// TIA Portal V17 export
// export: Created 2022-07-20T07:02:34.5888701Z, ExportSetting WithDefaults, DisplayName Totally Integrated Automation Portal, DisplayVersion V17, DisplayName TIA Portal Openness, DisplayVersion V17, DisplayName TIA Portal Version Control Interface, DisplayVersion V17, DisplayName SINAMICS Startdrive Advanced, DisplayVersion V17, DisplayName SINAMICS Startdrive G130, G150, S120, S150, SINAMICS MV, S210, DisplayVersion V17, DisplayName SINAMICS Startdrive G110M, G120, G120C, G120D, G120P, G115D, DisplayVersion V17, DisplayName STEP 7 Professional, DisplayVersion V17, DisplayName STEP 7 Safety, DisplayVersion V17, DisplayName WinCC Advanced, DisplayVersion V17
FUNCTION_BLOCK "FB10373_IOLinkConfig_Any"   // FB10373, LAD
{ S7_Optimized_Access := 'TRUE' }
VERSION : 0.1
// stored: AutoNumber false, IsIECCheckEnabled false, IsRetainMemResEnabled false, MemoryReserve 100, SetENOAutomatically false, UDAEnableTagReadback false
   VAR_INPUT
      Ackowledge : Bool;
      PortDevice : Int;
      Id : HW_IO;
      RequestGetParamID : Bool;
      RequestSetParamID : Bool;
      Index : Int;
      SubIndex : Int;
      Length : Int;
   END_VAR
   VAR_OUTPUT
      ParamIdDone : Bool;
      ParamConfigFault : Array[0..231] of Byte;
      Error : Bool;
      Status : Word;
   END_VAR
   VAR_IN_OUT
      Value : Array[0..231] of Byte;
   END_VAR
   VAR
      CommandStruct : Struct
         In : Struct
            TrigStart_Pulse : Bool;
            Id : HW_IO;
            rw : Bool;
            Port : Int;
            index : Int;
            subindex : Int;
            length : Int;
         END_STRUCT;
         Out : Struct
            Done : Bool;
            busy : Bool;
            Error : Bool;
            Status : Word;
         END_STRUCT;
         InOut : Struct
            Data : Array[0..231] of Byte;
         END_STRUCT;
      END_STRUCT;
      RequestPulseTrigStart : Bool;
      IoLinkConfigurationStateDiagram : Int;
      ParameterDone : Bool;
      R_TRIG_RequestGetParamId { S7_SetPoint := 'True'} : R_TRIG;
      R_TRIG_RequestSetParamId { S7_SetPoint := 'True'} : R_TRIG;
      FB10003_Pulse_Instance { S7_SetPoint := 'True'} : "FB10003_Pulse";
      FB10370_IoLinkDevice_Instance_1 { S7_SetPoint := 'True'} : "FB10370_IoLinkDevice";
   END_VAR
   VAR CONSTANT
      WAIT_FOR_IO_LINK_CONFIGURATION_COMMAND : Int := 0;
      RESTORE_DEFAULT_SETTINGS_IN_PROGRESS : Int := 10;
      GET_PARAM_ID_IN_PROGRESS : Int := 20;
      SET_PARAM_ID_IN_PROGRESS : Int := 30;
      READ_POWER_CYCLES_IN_PROGRESS : Int := 40;
      IO_LINK_COMMAND_CONFIGURATION_DONE : Int := 100;
      CAP_IO_LINK_IFM : Int := 19456;
   END_VAR
BEGIN

REGION Network 1 (SCL): First Scan
   IF "FirstScan" THEN
       #ParamIdDone := FALSE;
       #IoLinkConfigurationStateDiagram := #WAIT_FOR_IO_LINK_CONFIGURATION_COMMAND;
   END_IF;
END_REGION

REGION Network 2 (SCL): Edge Signals, Timers, Pulse
   REGION EDGE SIGNALS 
       #R_TRIG_RequestGetParamId(CLK := #RequestGetParamID);
       #R_TRIG_RequestSetParamId(CLK := #RequestSetParamID);

   END_REGION

   REGION TIMERS 

   END_REGION

   REGION PULSE
       #FB10003_Pulse_Instance(CLK := #RequestPulseTrigStart,
                               PT := T#50ms,
                               Q := #CommandStruct.In.TrigStart_Pulse);
   END_REGION
END_REGION

REGION Network 3 (SCL): Io Link Commands Management
   #CommandStruct.In.Port := #PortDevice;
   #CommandStruct.In.Id := #Id;
END_REGION

REGION Network 4: Io Link Configuration Manager
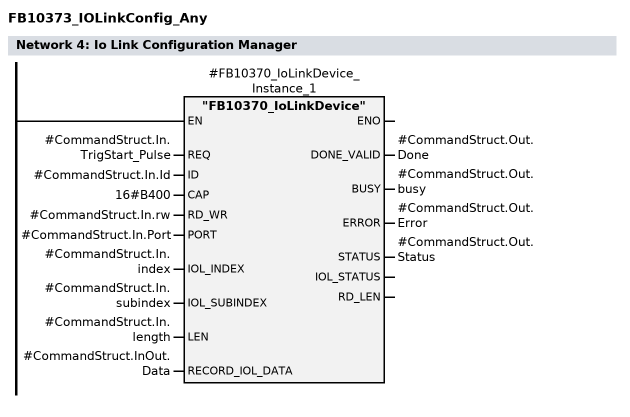
   RUNG wire#powerrail
      #FB10370_IoLinkDevice_Instance_1(REQ := #CommandStruct.In.TrigStart_Pulse, ID := #CommandStruct.In.Id, CAP := 16#B400, RD_WR := #CommandStruct.In.rw, PORT := #CommandStruct.In.Port, IOL_INDEX := #CommandStruct.In.index, IOL_SUBINDEX := #CommandStruct.In.subindex, LEN := #CommandStruct.In.length, RECORD_IOL_DATA := #CommandStruct.InOut.Data, DONE_VALID => #CommandStruct.Out.Done, BUSY => #CommandStruct.Out.busy, ERROR => #CommandStruct.Out.Error, STATUS => #CommandStruct.Out.Status, IOL_STATUS =>, RD_LEN =>)
   END_RUNG
   // the same network as SCL:
   #FB10370_IoLinkDevice_Instance_1(REQ := #CommandStruct.In.TrigStart_Pulse,   // "FB10370_IoLinkDevice"
                           ID := #CommandStruct.In.Id,
                           CAP := 16#B400,
                           RD_WR := #CommandStruct.In.rw,
                           PORT := #CommandStruct.In.Port,
                           IOL_INDEX := #CommandStruct.In.index,
                           IOL_SUBINDEX := #CommandStruct.In.subindex,
                           LEN := #CommandStruct.In.length,
                           RECORD_IOL_DATA := #CommandStruct.InOut.Data,
                           DONE_VALID => #CommandStruct.Out.Done,
                           BUSY => #CommandStruct.Out.busy,
                           ERROR => #CommandStruct.Out.Error,
                           STATUS => #CommandStruct.Out.Status);
END_REGION

REGION Network 5 (SCL): Io Link Commands Configuration Management
   CASE #IoLinkConfigurationStateDiagram OF

       #WAIT_FOR_IO_LINK_CONFIGURATION_COMMAND:
           IF #R_TRIG_RequestGetParamId.Q THEN
               #ParamIdDone := FALSE;
               #CommandStruct.In.index := #Index;
               #CommandStruct.In.subindex := #SubIndex;
               #CommandStruct.In.rw := FALSE;
               #CommandStruct.In.length := #Length;

               #Value := #CommandStruct.InOut.Data;
               #IoLinkConfigurationStateDiagram := #GET_PARAM_ID_IN_PROGRESS;

           ELSIF #R_TRIG_RequestSetParamId.Q THEN
               #ParamIdDone := FALSE;
               #CommandStruct.InOut.Data := #Value;
               #CommandStruct.In.index := #Index;
               #CommandStruct.In.subindex := #SubIndex;
               #CommandStruct.In.rw := TRUE;
               #CommandStruct.In.length := #Length;
               #IoLinkConfigurationStateDiagram := #SET_PARAM_ID_IN_PROGRESS;
           END_IF;


       #GET_PARAM_ID_IN_PROGRESS:
           REGION State Action Management
               #RequestPulseTrigStart := TRUE;
              // #CommandStruct.In.Data := #SP1_Value;
           END_REGION

           REGION State Exit Management
               IF #CommandStruct.Out.Done THEN
                   #ParamIdDone := TRUE;
                   #RequestPulseTrigStart := FALSE;
                   #IoLinkConfigurationStateDiagram := #IO_LINK_COMMAND_CONFIGURATION_DONE;
               END_IF;
           END_REGION

       #SET_PARAM_ID_IN_PROGRESS:
           REGION State Action Management
               #RequestPulseTrigStart := TRUE;
               // #CommandStruct.In.Data := #SP1_Value;
           END_REGION

           REGION State Exit Management
               IF #CommandStruct.Out.Done THEN
                   #ParamIdDone := TRUE;
                   #RequestPulseTrigStart := FALSE;
                   #IoLinkConfigurationStateDiagram := #IO_LINK_COMMAND_CONFIGURATION_DONE;
               END_IF;
           END_REGION


       #IO_LINK_COMMAND_CONFIGURATION_DONE:
           #ParameterDone := FALSE;
           #IoLinkConfigurationStateDiagram := #WAIT_FOR_IO_LINK_CONFIGURATION_COMMAND;
   END_CASE;
END_REGION

REGION Network 6 (SCL): Io Link Commands Error Management
   IF #CommandStruct.Out.Error THEN
       #IoLinkConfigurationStateDiagram := #WAIT_FOR_IO_LINK_CONFIGURATION_COMMAND;
       #Error := TRUE;
   END_IF;

   IF #Ackowledge THEN
       #Error := FALSE;
   END_IF;
   #Status := #CommandStruct.Out.Status;
END_REGION
END_FUNCTION_BLOCK
